TYPE "PLCtoMES_MainCheckOut"
VERSION : 0.1
   STRUCT
      "P-DataSaveReq" : Bool;
      "P-PartType" : String[28];
      "P-PartID" : Array[1..10] of String[48];
      "P-SubPartID" : Array[1..10] of String[48];
      "P-PartResult" : Byte;
      "P-RecipeVer" : String[18];
      Reserve : Array[1..1146] of Byte;
   END_STRUCT;

END_TYPE

